(* CODESYS project Untitled1.project

Project tree, tasks and I/O mapping:
  Device : CODESYS Control Win V3, 3S - Smart Software Solutions GmbH, order no. 305021, version 3.5.11.30
    application Application
      libraries: Standard, * (System)
      task MainTask (cyclic, interval t#20ms, priority 1) calls PLC_PRG
      program PLC_PRG [SFC]: P2_entry, TS1, P2_active
*)

// Device/Application/PLC_PRG
PROGRAM PLC_PRG
VAR
	B1: BOOL;
	KM1: BOOL;
	S1: BOOL;
	YA: BOOL;
	Trans1: BOOL;
	CT1:INT;
	YC: BOOL;
	YB: BOOL;
	RT1: R_TRIG;
END_VAR

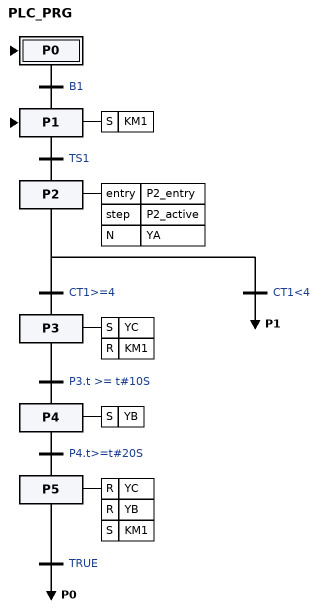
INITIAL_STEP P0:
END_STEP
TRANSITION FROM P0 TO P1
    := B1;
END_TRANSITION
STEP P1:
    KM1(S);
END_STEP
TRANSITION FROM P1 TO P2
    := TS1;
END_TRANSITION
STEP P2:
    P2_entry(P1);  // entry action
    P2_active(N);  // step action
    YA(N);
END_STEP
TRANSITION FROM P2 TO P3
    := CT1>=4;
END_TRANSITION
STEP P3:
    YC(S);
    KM1(R);
END_STEP
TRANSITION FROM P2 TO P1
    := CT1<4;
END_TRANSITION
TRANSITION FROM P3 TO P4
    := P3.t >= t#10S;
END_TRANSITION
STEP P4:
    YB(S);
END_STEP
TRANSITION FROM P4 TO P5
    := P4.t>=t#20S;
END_TRANSITION
STEP P5:
    YC(R);
    YB(R);
    KM1(S);
END_STEP
TRANSITION FROM P5 TO P0
    := TRUE;
END_TRANSITION

ACTION P2_entry:
CT1:= CT1 + 1;
END_ACTION

TRANSITION TS1:
RT1(CLK:=S1);

IF RT1.Q THEN
	TS1:= TRUE;
	ELSE
		TS1:= FALSE;
END_IF
END_TRANSITION

ACTION P2_active:

END_ACTION

END_PROGRAM
